// TIA Portal project "sıralı_lamba" (V18)

(* hardware
DEVICE "S7-1200 station_1"  S7-1200 Station
   slot 0: "Rack_0"  S7-1200 Rack  Rack  V1.0
   slot 1: "PLC_1"  CPU 1212C DC/DC/DC  6ES7 212-1AE40-0XB0  V4.6
*)

// ===== PLC "PLC_1"  CPU 1212C DC/DC/DC =====

VAR_GLOBAL   // PLC tag table "Default tag table"
   "BUTON" AT %I0.0 : Bool;
   "A" AT %M0.0 : Bool;
   "B" AT %M0.1 : Bool;
   "C" AT %M0.2 : Bool;
   "D" AT %M0.3 : Bool;
   "X" AT %M10.0 : Bool;
   "E" AT %M0.4 : Bool;
   "F" AT %M0.5 : Bool;
   "G" AT %M0.6 : Bool;
   "H" AT %M0.7 : Bool;
   "L1" AT %Q1.0 : Bool;
   "L2" AT %Q1.1 : Bool;
   "L3" AT %Q1.2 : Bool;
   "L4" AT %Q1.3 : Bool;
   "TPOUT" AT %M2.0 : Bool;
   "CTUOUT" AT %M2.1 : Bool;
   "CMPOUT" AT %M2.2 : Bool;
   "BTN" AT %M2.3 : Bool;
   "I" AT %M3.0 : Bool;
   "J" AT %M3.1 : Bool;
   "K" AT %M3.2 : Bool;
   "L" AT %M3.3 : Bool;
   "Tag_1" AT %M2.4 : Bool;
END_VAR

// folder: System blocks/Program resources

DATA_BLOCK "IEC_Timer_0_DB"   // DB1
{ S7_Optimized_Access := 'TRUE' }
AUTHOR : Simatic
FAMILY : IEC
NAME : IEC_TMR
VERSION : 1.0
// stored: InstanceOfName IEC_TIMER
"IEC_TIMER"
BEGIN
END_DATA_BLOCK

DATA_BLOCK "IEC_Counter_0_DB_1"   // DB4
{ S7_Optimized_Access := 'TRUE' }
AUTHOR : Simatic
FAMILY : IEC
NAME : CNTR
VERSION : 1.0
// stored: InstanceOfName IEC_COUNTER
"IEC_COUNTER"
BEGIN
END_DATA_BLOCK

// folder: (top level)

FUNCTION "Block_1" : Void   // FC1, LAD
{ S7_Optimized_Access := 'TRUE' }
VERSION : 0.1
BEGIN

REGION Network 1
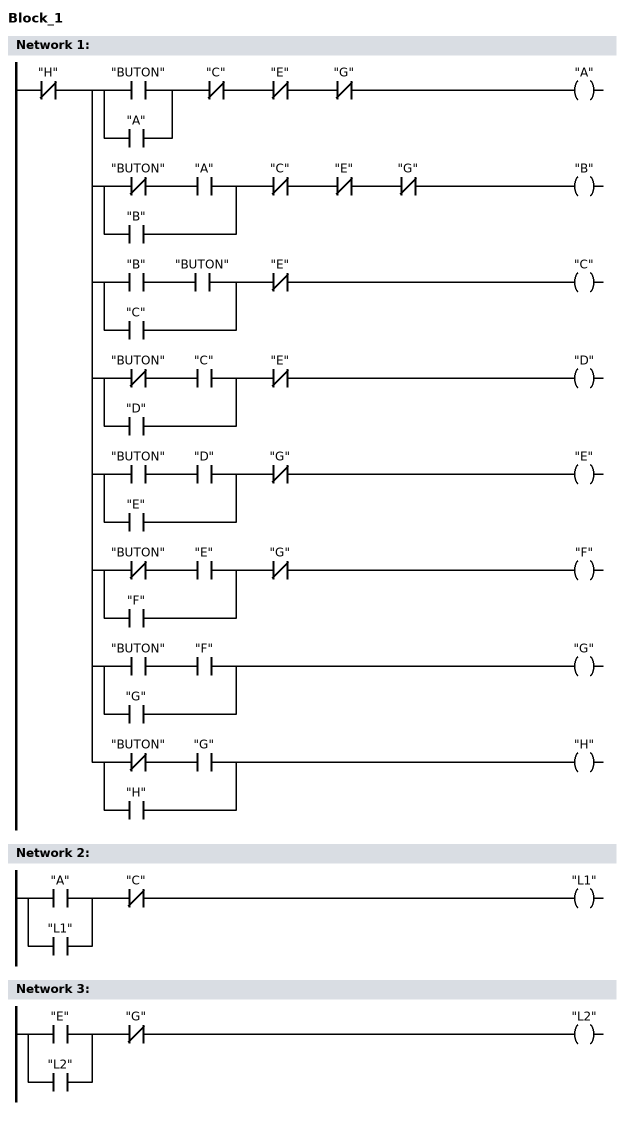
   RUNG wire#powerrail
      I_Contact( "H" )
      wire#w1
      Contact( "BUTON" )
      wire#w2
      I_Contact( "C" )
      I_Contact( "E" )
      I_Contact( "G" )
      Coil( "A" )
   END_RUNG
   RUNG wire#w1
      Contact( "A" )
   END_RUNG wire#w2
   RUNG wire#w1
      I_Contact( "BUTON" )
      Contact( "A" )
      wire#w3
      I_Contact( "C" )
      I_Contact( "E" )
      I_Contact( "G" )
      Coil( "B" )
   END_RUNG
   RUNG wire#w1
      Contact( "B" )
   END_RUNG wire#w3
   RUNG wire#w1
      Contact( "B" )
      Contact( "BUTON" )
      wire#w4
      I_Contact( "E" )
      Coil( "C" )
   END_RUNG
   RUNG wire#w1
      Contact( "C" )
   END_RUNG wire#w4
   RUNG wire#w1
      I_Contact( "BUTON" )
      Contact( "C" )
      wire#w5
      I_Contact( "E" )
      Coil( "D" )
   END_RUNG
   RUNG wire#w1
      Contact( "D" )
   END_RUNG wire#w5
   RUNG wire#w1
      Contact( "BUTON" )
      Contact( "D" )
      wire#w6
      I_Contact( "G" )
      Coil( "E" )
   END_RUNG
   RUNG wire#w1
      Contact( "E" )
   END_RUNG wire#w6
   RUNG wire#w1
      I_Contact( "BUTON" )
      Contact( "E" )
      wire#w7
      I_Contact( "G" )
      Coil( "F" )
   END_RUNG
   RUNG wire#w1
      Contact( "F" )
   END_RUNG wire#w7
   RUNG wire#w1
      Contact( "BUTON" )
      Contact( "F" )
      wire#w8
      Coil( "G" )
   END_RUNG
   RUNG wire#w1
      Contact( "G" )
   END_RUNG wire#w8
   RUNG wire#w1
      I_Contact( "BUTON" )
      Contact( "G" )
      wire#w9
      Coil( "H" )
   END_RUNG
   RUNG wire#w1
      Contact( "H" )
   END_RUNG wire#w9
   // the same network as SCL:
   "A" := NOT "H" AND ("BUTON" OR "A") AND NOT "C" AND NOT "E" AND NOT "G";
   "B" := NOT "H" AND ((NOT "BUTON" AND "A") OR "B") AND NOT "C" AND NOT "E" AND NOT "G";
   "C" := NOT "H" AND (("B" AND "BUTON") OR "C") AND NOT "E";
   "D" := NOT "H" AND ((NOT "BUTON" AND "C") OR "D") AND NOT "E";
   "E" := NOT "H" AND (("BUTON" AND "D") OR "E") AND NOT "G";
   "F" := NOT "H" AND ((NOT "BUTON" AND "E") OR "F") AND NOT "G";
   "G" := NOT "H" AND (("BUTON" AND "F") OR "G");
   "H" := NOT "H" AND ((NOT "BUTON" AND "G") OR "H");
END_REGION

REGION Network 2
   RUNG wire#powerrail
      Contact( "A" )
      wire#w1
      I_Contact( "C" )
      Coil( "L1" )
   END_RUNG
   RUNG wire#powerrail
      Contact( "L1" )
   END_RUNG wire#w1
   // the same network as SCL:
   "L1" := ("A" OR "L1") AND NOT "C";
END_REGION

REGION Network 3
   RUNG wire#powerrail
      Contact( "E" )
      wire#w1
      I_Contact( "G" )
      Coil( "L2" )
   END_RUNG
   RUNG wire#powerrail
      Contact( "L2" )
   END_RUNG wire#w1
   // the same network as SCL:
   "L2" := ("E" OR "L2") AND NOT "G";
END_REGION
END_FUNCTION

FUNCTION "timer" : Void   // FC2, LAD
{ S7_Optimized_Access := 'TRUE' }
VERSION : 0.1
   VAR_TEMP   // added for the SCL form of the ladder/FBD networks
      _w1 : Bool;
   END_VAR
BEGIN

REGION Network 1
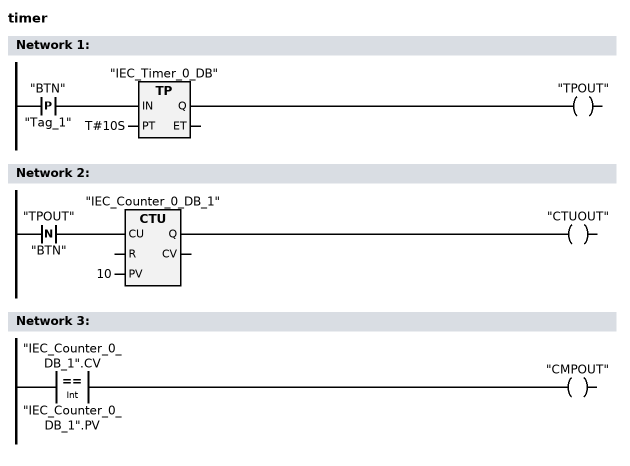
   #_w1 := "BTN" AND NOT "Tag_1";   // rising edge of "BTN"
   "Tag_1" := "BTN";
   "IEC_Timer_0_DB".TP(IN := #_w1, PT := T#10S);
   "TPOUT" := "IEC_Timer_0_DB".Q;
END_REGION

REGION Network 2
   #_w1 := NOT "TPOUT" AND "BTN";   // falling edge of "TPOUT"
   "BTN" := "TPOUT";
   "IEC_Counter_0_DB_1".CTU(CU := #_w1, PV := 10);
   "CTUOUT" := "IEC_Counter_0_DB_1".Q;
END_REGION

REGION Network 3
   RUNG wire#powerrail
      { S7_Templates := "SrcType := Int" } EQ_Contact(in1 := "IEC_Counter_0_DB_1".CV, in2 := "IEC_Counter_0_DB_1".PV)
      Coil( "CMPOUT" )
   END_RUNG
   // the same network as SCL:
   "CMPOUT" := "IEC_Counter_0_DB_1".CV = "IEC_Counter_0_DB_1".PV;
END_REGION
END_FUNCTION

FUNCTION "Block_2" : Void   // FC3, LAD
{ S7_Optimized_Access := 'TRUE' }
VERSION : 0.1
BEGIN

REGION Network 1
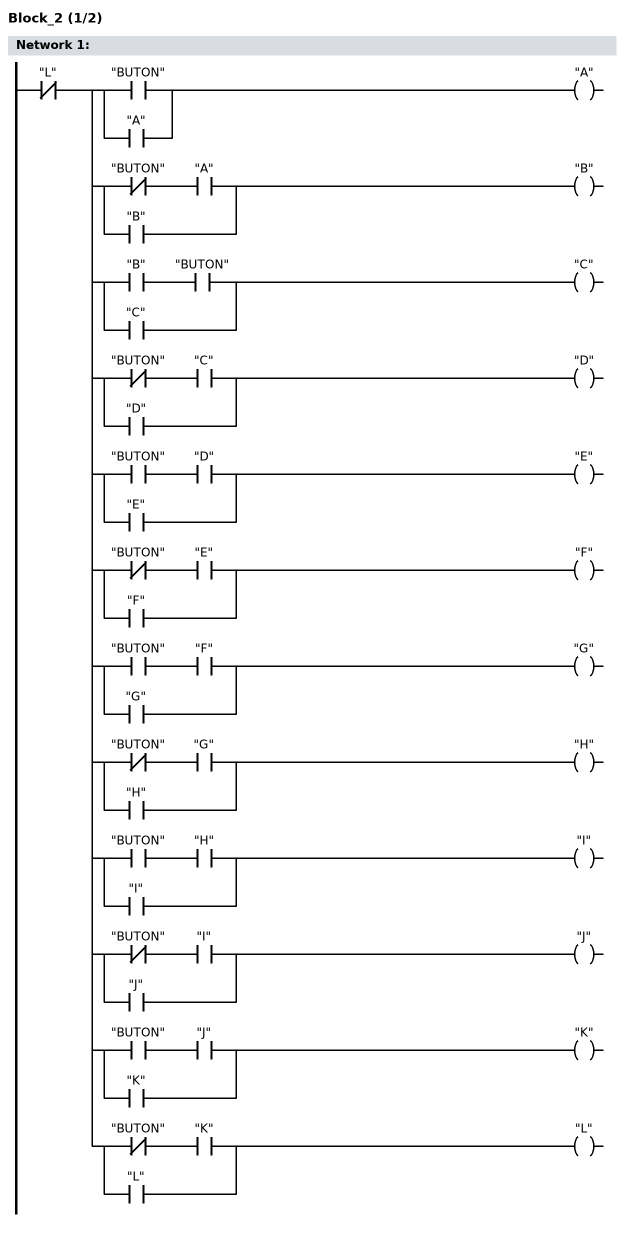
   RUNG wire#powerrail
      I_Contact( "L" )
      wire#w1
      Contact( "BUTON" )
      wire#w2
      Coil( "A" )
   END_RUNG
   RUNG wire#w1
      Contact( "A" )
   END_RUNG wire#w2
   RUNG wire#w1
      I_Contact( "BUTON" )
      Contact( "A" )
      wire#w3
      Coil( "B" )
   END_RUNG
   RUNG wire#w1
      Contact( "B" )
   END_RUNG wire#w3
   RUNG wire#w1
      Contact( "B" )
      Contact( "BUTON" )
      wire#w4
      Coil( "C" )
   END_RUNG
   RUNG wire#w1
      Contact( "C" )
   END_RUNG wire#w4
   RUNG wire#w1
      I_Contact( "BUTON" )
      Contact( "C" )
      wire#w5
      Coil( "D" )
   END_RUNG
   RUNG wire#w1
      Contact( "D" )
   END_RUNG wire#w5
   RUNG wire#w1
      Contact( "BUTON" )
      Contact( "D" )
      wire#w6
      Coil( "E" )
   END_RUNG
   RUNG wire#w1
      Contact( "E" )
   END_RUNG wire#w6
   RUNG wire#w1
      I_Contact( "BUTON" )
      Contact( "E" )
      wire#w7
      Coil( "F" )
   END_RUNG
   RUNG wire#w1
      Contact( "F" )
   END_RUNG wire#w7
   RUNG wire#w1
      Contact( "BUTON" )
      Contact( "F" )
      wire#w8
      Coil( "G" )
   END_RUNG
   RUNG wire#w1
      Contact( "G" )
   END_RUNG wire#w8
   RUNG wire#w1
      I_Contact( "BUTON" )
      Contact( "G" )
      wire#w9
      Coil( "H" )
   END_RUNG
   RUNG wire#w1
      Contact( "H" )
   END_RUNG wire#w9
   RUNG wire#w1
      Contact( "BUTON" )
      Contact( "H" )
      wire#w10
      Coil( "I" )
   END_RUNG
   RUNG wire#w1
      Contact( "I" )
   END_RUNG wire#w10
   RUNG wire#w1
      I_Contact( "BUTON" )
      Contact( "I" )
      wire#w11
      Coil( "J" )
   END_RUNG
   RUNG wire#w1
      Contact( "J" )
   END_RUNG wire#w11
   RUNG wire#w1
      Contact( "BUTON" )
      Contact( "J" )
      wire#w12
      Coil( "K" )
   END_RUNG
   RUNG wire#w1
      Contact( "K" )
   END_RUNG wire#w12
   RUNG wire#w1
      I_Contact( "BUTON" )
      Contact( "K" )
      wire#w13
      Coil( "L" )
   END_RUNG
   RUNG wire#w1
      Contact( "L" )
   END_RUNG wire#w13
   // the same network as SCL:
   "A" := NOT "L" AND ("BUTON" OR "A");
   "B" := NOT "L" AND ((NOT "BUTON" AND "A") OR "B");
   "C" := NOT "L" AND (("B" AND "BUTON") OR "C");
   "D" := NOT "L" AND ((NOT "BUTON" AND "C") OR "D");
   "E" := NOT "L" AND (("BUTON" AND "D") OR "E");
   "F" := NOT "L" AND ((NOT "BUTON" AND "E") OR "F");
   "G" := NOT "L" AND (("BUTON" AND "F") OR "G");
   "H" := NOT "L" AND ((NOT "BUTON" AND "G") OR "H");
   "I" := NOT "L" AND (("BUTON" AND "H") OR "I");
   "J" := NOT "L" AND ((NOT "BUTON" AND "I") OR "J");
   "K" := NOT "L" AND (("BUTON" AND "J") OR "K");
   "L" := NOT "L" AND ((NOT "BUTON" AND "K") OR "L");
END_REGION

REGION Network 2
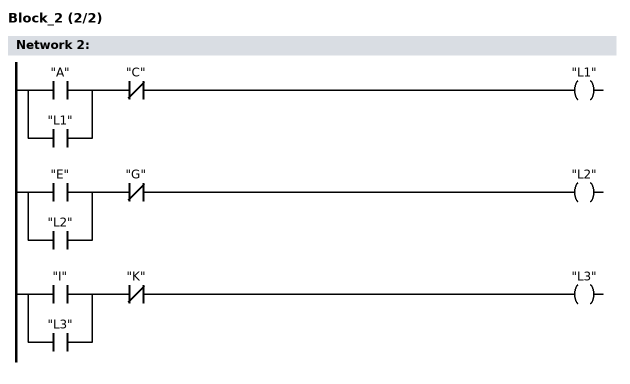
   RUNG wire#powerrail
      Contact( "A" )
      wire#w1
      I_Contact( "C" )
      Coil( "L1" )
   END_RUNG
   RUNG wire#powerrail
      Contact( "L1" )
   END_RUNG wire#w1
   RUNG wire#powerrail
      Contact( "E" )
      wire#w2
      I_Contact( "G" )
      Coil( "L2" )
   END_RUNG
   RUNG wire#powerrail
      Contact( "L2" )
   END_RUNG wire#w2
   RUNG wire#powerrail
      Contact( "I" )
      wire#w3
      I_Contact( "K" )
      Coil( "L3" )
   END_RUNG
   RUNG wire#powerrail
      Contact( "L3" )
   END_RUNG wire#w3
   // the same network as SCL:
   "L1" := ("A" OR "L1") AND NOT "C";
   "L2" := ("E" OR "L2") AND NOT "G";
   "L3" := ("I" OR "L3") AND NOT "K";
END_REGION
END_FUNCTION

ORGANIZATION_BLOCK "Main"   // OB1, LAD, ProgramCycle
TITLE = "Main Program Sweep (Cycle)"
{ S7_Optimized_Access := 'TRUE' }
VERSION : 0.1
   VAR_INPUT
      Initial_Call : Bool;   // Initial call of this OB
      Remanence : Bool;   // =True, if remanent data are available
   END_VAR
BEGIN

REGION Network 1
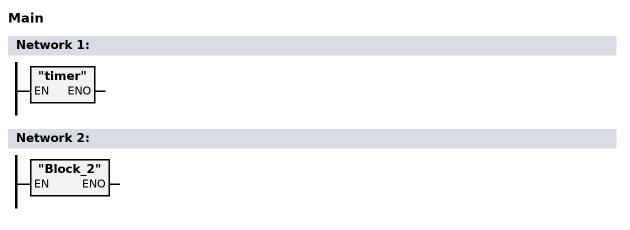
   RUNG wire#powerrail
      "timer"()
   END_RUNG
   // the same network as SCL:
   "timer"();
END_REGION

REGION Network 2
   RUNG wire#powerrail
      "Block_2"()
   END_RUNG
   // the same network as SCL:
   "Block_2"();
END_REGION
END_ORGANIZATION_BLOCK